{attribute addProperty BoxType "EP7402-0057-0017"}
{attribute addProperty Id "InputAT %I*ARRAY[0 ..3] OF BOOL3240Control_inputAT %I*ARRAY[0 ..3] OF BOOL3240"}
{attribute addProperty CRC "979228258"}
{attribute addProperty SizeInBites "64"}
{attribute addProperty SizeInBytes "8"}
TYPE DI_Inputs_3959EB25 :
STRUCT
	{attribute addProperty Name "Input"}
	Input AT %I* : ARRAY[0 ..3] OF BOOL;
	{attribute addProperty Name "Control_input"}
	Control_input AT %I* : ARRAY[0 ..3] OF BOOL;
END_STRUCT
END_TYPE

(* stored: Version 1.2.0.0, ProductVersion 3.1.4024.9
   DUT DI_Inputs_3959EB25: Id {cc6ad84c-ce1d-4b85-9ce4-6f7954d98e20} *)
